PROGRAM UnitTests
VAR
	fbTestRound		: Fb_TestRound;
	fbTestSplit		: FB_TestSplit;
END_VAR

TcUnit.RUN();

END_PROGRAM

(* stored: Version 1.1.0.1, ProductVersion 3.1.4024.9
   POU UnitTests: Id {6e2183c7-16a4-43f8-8211-71db06d79010}, SpecialFunc None *)
